Universal Robots PolyScope program: move.urp

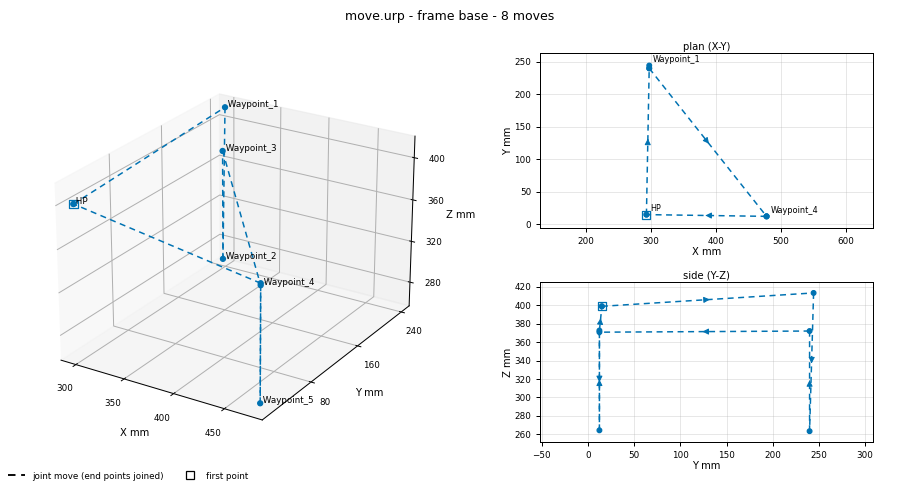
[picture p0: tool path of move.urp in frame base, 8 of 8 moves have a stored position in this frame; points joined in program order, loops and branches not executed]
Program move (installation=default directory=/programs/palletizing createdIn=5.11.9.1010452 lastSavedIn=5.11.9.1010452 robotSerialNumber=20225200364)
Calibrated DH parameters: a=[0.00002, -0.569483, -0.54992, -0.00001, -0.000036, 0]; d=[0.180894, -146.691669, 192.918669, -46.053088, 0.119778, 0.115602]; alpha=[1.571425, -0.001534, 0.003359, 1.568739, -1.571477, 0]; deltaTheta=[0, 0.376258, -0.101074, -0.275185, -0.000002, 0]
Robot Program (runOnlyOnce=false)
  URCap RG Grip (OnRobot, OnRobot A/S) dataModel(rg-target-force=40.0, rg-target-width=0.1, Variable(key=on_return, variable(name=on_return)))
  MoveJ speed 60 deg/s, acceleration 80 deg/s^2 (useActiveTCP=true) feature=Base
    Waypoint HP: TCP in base x=293 y=15.068 z=398.718 mm, rx=2.2313 ry=-2.2053 rz=0.0033 rad; joints [39.469, -75.55, -131.598, -243.13, -90.057, -140.975] deg
    Waypoint Waypoint_1: TCP in base x=297.33 y=244.272 z=413.188 mm, rx=2.2312 ry=-2.2053 rz=0.0033 rad; joints [66.332, -85.91, -121.62, -242.789, -90.169, -114.102] deg
    Waypoint Waypoint_2: TCP in base x=297.313 y=239.934 z=263.51 mm, rx=2.2042 ry=-2.2324 rz=0.0035 rad; joints [66.068, -95.967, -130.16, -224.192, -90.128, -112.905] deg
    URCap RG Grip (OnRobot, OnRobot A/S) dataModel(rg-target-force=40.0, rg-target-width=0.075)
    Waypoint Waypoint_3: TCP in base x=297.333 y=239.94 z=371.956 mm, rx=2.2041 ry=-2.2325 rz=0.0035 rad; joints [66.048, -87.905, -124.53, -237.883, -90.158, -112.967] deg
    Waypoint Waypoint_4: TCP in base x=477.669 y=12.407 z=370.707 mm, rx=2.1969 ry=-2.2396 rz=0.0034 rad; joints [22.917, -97.492, -114.493, -238.242, -89.962, -155.725] deg
    Waypoint Waypoint_5: TCP in base x=477.679 y=12.404 z=264.445 mm, rx=2.1969 ry=-2.2396 rz=0.0034 rad; joints [22.925, -104.326, -119.411, -226.49, -89.937, -155.678] deg
    URCap RG Grip (OnRobot, OnRobot A/S) dataModel(rg-target-force=40.0, rg-target-width=0.1)
    Waypoint Waypoint_6: TCP in base x=477.682 y=12.403 z=372.508 mm, rx=2.1969 ry=-2.2396 rz=0.0034 rad; joints [22.915, -97.396, -114.392, -238.441, -89.964, -155.726] deg
    Waypoint Waypoint_7: TCP in base x=293.016 y=15.071 z=398.727 mm, rx=2.2313 ry=-2.2054 rz=0.0034 rad; joints [39.467, -75.549, -131.596, -243.126, -90.057, -140.975] deg
    Halt
